(* CODESYS project TrabalhoFMSSFC.project

Project tree, tasks and I/O mapping:
  Device : CODESYS Control Win V3, 3S - Smart Software Solutions GmbH, order no. 305021, version 3.5.11.30
    application Application
      libraries: Standard, * (System)
      task MainTask (cyclic, interval t#20ms, priority 1) calls Inicializacao
      program Inicializacao [SFC]
      program estacaoPallet [SFC]
      program SaidaPecas [SFC]
      program esteira [SFC]
      program RobosDaora [SFC]
      program EstacaoTampa [SFC]
      program Armazenamento [SFC]
  program Inicializacao [SFC]
  program POU [CFC]
*)

// Device/Application/Inicializacao
PROGRAM Inicializacao
VAR
	Bot: INT;
	o_lig: INT;
	o_off: INT;
	o_On: INT;
	Botao_on: BOOL;
	Botao_off: BOOL;
END_VAR

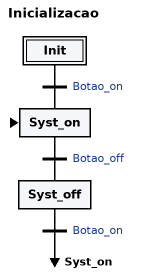
INITIAL_STEP Init:
END_STEP
TRANSITION FROM Init TO Syst_on
    := Botao_on;
END_TRANSITION
STEP Syst_on:
END_STEP
TRANSITION FROM Syst_on TO Syst_off
    := Botao_off;
END_TRANSITION
STEP Syst_off:
END_STEP
TRANSITION FROM Syst_off TO Syst_on
    := Botao_on;
END_TRANSITION

END_PROGRAM

// Inicializacao
PROGRAM Inicializacao
VAR
	Bot: INT;
	o_lig: INT;
	o_off: INT;
	o_On: INT;
	Botao_on: BOOL;
	Botao_off: BOOL;
END_VAR

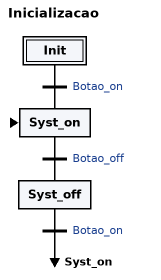
INITIAL_STEP Init:
END_STEP
TRANSITION FROM Init TO Syst_on
    := Botao_on;
END_TRANSITION
STEP Syst_on:
END_STEP
TRANSITION FROM Syst_on TO Syst_off
    := Botao_off;
END_TRANSITION
STEP Syst_off:
END_STEP
TRANSITION FROM Syst_off TO Syst_on
    := Botao_on;
END_TRANSITION

END_PROGRAM

// Device/Application/estacaoPallet
PROGRAM estacaoPallet
VAR_INPUT
END_VAR
VAR_OUTPUT
END_VAR
VAR
	Sistema_on: BOOL;
	diffuse_sensor_3_clp: BOOL;
	diffuse_sensor_4_clp: BOOL;
	timer_1: BOOL;
	timer_2: BOOL;
	timer_3: BOOL;
	timer_5: BOOL;
	timer_6: BOOL;
	timer_7: BOOL;
	timer_8: BOOL;
	timer_9: BOOL;
END_VAR

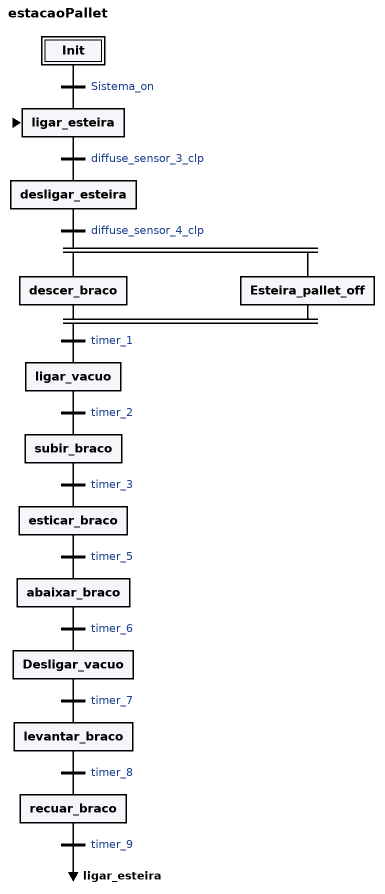
INITIAL_STEP Init:
END_STEP
TRANSITION FROM Init TO ligar_esteira
    := Sistema_on;
END_TRANSITION
STEP ligar_esteira:
END_STEP
TRANSITION FROM ligar_esteira TO desligar_esteira
    := diffuse_sensor_3_clp;
END_TRANSITION
STEP desligar_esteira:
END_STEP
TRANSITION FROM desligar_esteira TO (descer_braco, Esteira_pallet_off)
    := diffuse_sensor_4_clp;
END_TRANSITION
STEP descer_braco:
END_STEP
STEP Esteira_pallet_off:
END_STEP
TRANSITION FROM (descer_braco, Esteira_pallet_off) TO ligar_vacuo
    := timer_1;
END_TRANSITION
STEP ligar_vacuo:
END_STEP
TRANSITION FROM ligar_vacuo TO subir_braco
    := timer_2;
END_TRANSITION
STEP subir_braco:
END_STEP
TRANSITION FROM subir_braco TO esticar_braco
    := timer_3;
END_TRANSITION
STEP esticar_braco:
END_STEP
TRANSITION FROM esticar_braco TO abaixar_braco
    := timer_5;
END_TRANSITION
STEP abaixar_braco:
END_STEP
TRANSITION FROM abaixar_braco TO Desligar_vacuo
    := timer_6;
END_TRANSITION
STEP Desligar_vacuo:
END_STEP
TRANSITION FROM Desligar_vacuo TO levantar_braco
    := timer_7;
END_TRANSITION
STEP levantar_braco:
END_STEP
TRANSITION FROM levantar_braco TO recuar_braco
    := timer_8;
END_TRANSITION
STEP recuar_braco:
END_STEP
TRANSITION FROM recuar_braco TO ligar_esteira
    := timer_9;
END_TRANSITION

END_PROGRAM

// POU
PROGRAM POU
VAR
END_VAR

END_PROGRAM

// Device/Application/SaidaPecas
PROGRAM SaidaPecas
VAR
	Sist_on: BOOL;
	sensor_back: BOOL;
	sensor_front: BOOL;
	azul: BOOL;
	timer_1: BOOL;
	timer_2: BOOL;
	nao_azul: BOOL;
	zera_azul: BOOL;
END_VAR

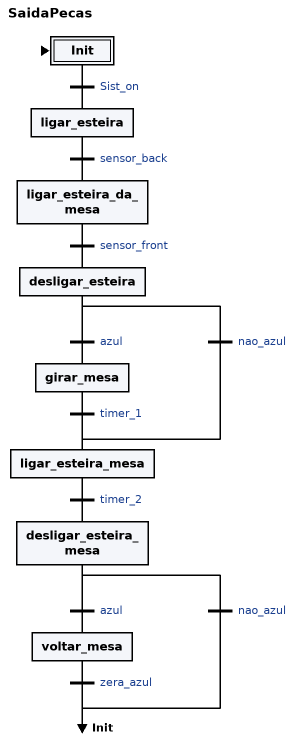
INITIAL_STEP Init:
END_STEP
TRANSITION FROM Init TO ligar_esteira
    := Sist_on;
END_TRANSITION
STEP ligar_esteira:
END_STEP
TRANSITION FROM ligar_esteira TO ligar_esteira_da_mesa
    := sensor_back;
END_TRANSITION
STEP ligar_esteira_da_mesa:
END_STEP
TRANSITION FROM ligar_esteira_da_mesa TO desligar_esteira
    := sensor_front;
END_TRANSITION
STEP desligar_esteira:
END_STEP
TRANSITION FROM desligar_esteira TO girar_mesa
    := azul;
END_TRANSITION
STEP girar_mesa:
END_STEP
TRANSITION FROM girar_mesa TO ligar_esteira_mesa
    := timer_1;
END_TRANSITION
TRANSITION FROM desligar_esteira TO ligar_esteira_mesa
    := nao_azul;
END_TRANSITION
STEP ligar_esteira_mesa:
END_STEP
TRANSITION FROM ligar_esteira_mesa TO desligar_esteira_mesa
    := timer_2;
END_TRANSITION
STEP desligar_esteira_mesa:
END_STEP
TRANSITION FROM desligar_esteira_mesa TO voltar_mesa
    := azul;
END_TRANSITION
STEP voltar_mesa:
END_STEP
TRANSITION FROM voltar_mesa TO Init
    := zera_azul;
END_TRANSITION
TRANSITION FROM desligar_esteira_mesa TO Init
    := nao_azul;
END_TRANSITION

END_PROGRAM

// Device/Application/esteira
PROGRAM esteira
VAR
	Bot: INT;
	o_lig: INT;
	o_off: INT;
	o_On: INT;
	Botao_on: BOOL;
	Botao_off: BOOL;
	Sensor_on: BOOL;
	Sensor_pff: BOOL;
	Sensor_off: BOOL;
	Sensor_Dif: BOOL;
	Sensor_Verde_on: BOOL;
	Sensor_Verde_off: BOOL;
	Timer_on: BOOL;
	Timer1_off: BOOL;
	Timer1_on: BOOL;
	Reset_Blade: BOOL;
	Sensor_presenca: BOOL;
	Sensor_Dif_on: BOOL;
	Sensor_Dif_off: BOOL;
	End_Blade: BOOL;
	Sensor_Dif1_on: BOOL;
	Sensor_Dif1_off: BOOL;
END_VAR

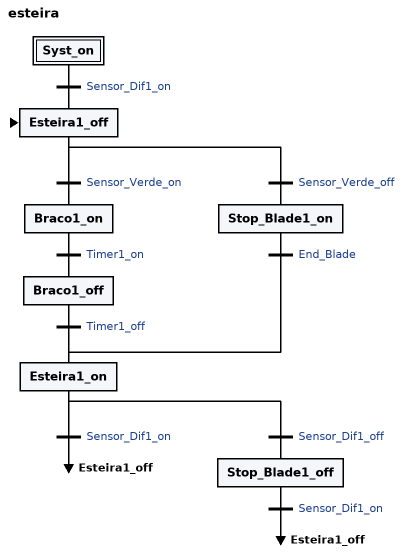
INITIAL_STEP Syst_on:
END_STEP
TRANSITION FROM Syst_on TO Esteira1_off
    := Sensor_Dif1_on;
END_TRANSITION
STEP Esteira1_off:
END_STEP
TRANSITION FROM Esteira1_off TO Braco1_on
    := Sensor_Verde_on;
END_TRANSITION
STEP Braco1_on:
END_STEP
TRANSITION FROM Braco1_on TO Braco1_off
    := Timer1_on;
END_TRANSITION
STEP Braco1_off:
END_STEP
TRANSITION FROM Braco1_off TO Esteira1_on
    := Timer1_off;
END_TRANSITION
TRANSITION FROM Esteira1_off TO Stop_Blade1_on
    := Sensor_Verde_off;
END_TRANSITION
STEP Stop_Blade1_on:
END_STEP
TRANSITION FROM Stop_Blade1_on TO Esteira1_on
    := End_Blade;
END_TRANSITION
STEP Esteira1_on:
END_STEP
TRANSITION FROM Esteira1_on TO Esteira1_off
    := Sensor_Dif1_on;
END_TRANSITION
TRANSITION FROM Esteira1_on TO Stop_Blade1_off
    := Sensor_Dif1_off;
END_TRANSITION
STEP Stop_Blade1_off:
END_STEP
TRANSITION FROM Stop_Blade1_off TO Esteira1_off
    := Sensor_Dif1_on;
END_TRANSITION

END_PROGRAM

// Device/Application/RobosDaora
PROGRAM RobosDaora
VAR
	Bot: INT;
	o_lig: INT;
	o_off: INT;
	o_On: INT;
	Botao_on: BOOL;
	Botao_off: BOOL;
	Robo1_Sens: BOOL;
	Robo1_Sens_on: BOOL;
	Robo1_end: BOOL;
END_VAR

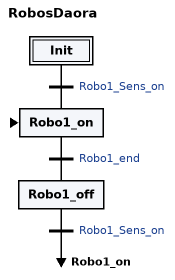
INITIAL_STEP Init:
END_STEP
TRANSITION FROM Init TO Robo1_on
    := Robo1_Sens_on;
END_TRANSITION
STEP Robo1_on:
END_STEP
TRANSITION FROM Robo1_on TO Robo1_off
    := Robo1_end;
END_TRANSITION
STEP Robo1_off:
END_STEP
TRANSITION FROM Robo1_off TO Robo1_on
    := Robo1_Sens_on;
END_TRANSITION

END_PROGRAM

// Device/Application/EstacaoTampa
PROGRAM EstacaoTampa
VAR
	//Entradas
	VisionSensor4_1:BOOL;
	VisionSensor4_0:BOOL;
	VIsionSensor4_2:BOOL;
	//SAIDAS
	Conveyor2m3:BOOL;
	PosicaoPegar: BOOL;
	ZPosition: BOOL;
	BoxDetected: BOOL;
	Grabber: BOOL;
	TampaPega: BOOL;
	Timer1: BOOL;
	Timer2: BOOL;
	PosicaoTampar: BOOL;
	Timer3: BOOL;
	Timer4: BOOL;
	Timer5: BOOL;
	StopBlade: BOOL;
	VisionSensor4_1Negado: BOOL;
END_VAR

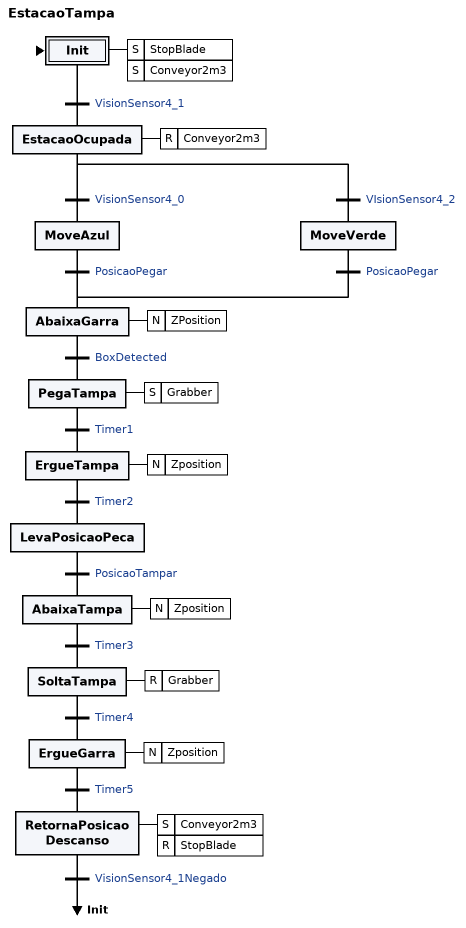
INITIAL_STEP Init:
    StopBlade(S);
    Conveyor2m3(S);
END_STEP
TRANSITION FROM Init TO EstacaoOcupada
    := VisionSensor4_1;
END_TRANSITION
STEP EstacaoOcupada:
    Conveyor2m3(R);
END_STEP
TRANSITION FROM EstacaoOcupada TO MoveAzul
    := VisionSensor4_0;
END_TRANSITION
STEP MoveAzul:
END_STEP
TRANSITION FROM MoveAzul TO AbaixaGarra
    := PosicaoPegar;
END_TRANSITION
TRANSITION FROM EstacaoOcupada TO MoveVerde
    := VIsionSensor4_2;
END_TRANSITION
STEP MoveVerde:
END_STEP
TRANSITION FROM MoveVerde TO AbaixaGarra
    := PosicaoPegar;
END_TRANSITION
STEP AbaixaGarra:
    ZPosition(N);
END_STEP
TRANSITION FROM AbaixaGarra TO PegaTampa
    := BoxDetected;
END_TRANSITION
STEP PegaTampa:
    Grabber(S);
END_STEP
TRANSITION FROM PegaTampa TO ErgueTampa
    := Timer1;
END_TRANSITION
STEP ErgueTampa:
    Zposition(N);
END_STEP
TRANSITION FROM ErgueTampa TO LevaPosicaoPeca
    := Timer2;
END_TRANSITION
STEP LevaPosicaoPeca:
END_STEP
TRANSITION FROM LevaPosicaoPeca TO AbaixaTampa
    := PosicaoTampar;
END_TRANSITION
STEP AbaixaTampa:
    Zposition(N);
END_STEP
TRANSITION FROM AbaixaTampa TO SoltaTampa
    := Timer3;
END_TRANSITION
STEP SoltaTampa:
    Grabber(R);
END_STEP
TRANSITION FROM SoltaTampa TO ErgueGarra
    := Timer4;
END_TRANSITION
STEP ErgueGarra:
    Zposition(N);
END_STEP
TRANSITION FROM ErgueGarra TO RetornaPosicaoDescanso
    := Timer5;
END_TRANSITION
STEP RetornaPosicaoDescanso:
    Conveyor2m3(S);
    StopBlade(R);
END_STEP
TRANSITION FROM RetornaPosicaoDescanso TO Init
    := VisionSensor4_1Negado;
END_TRANSITION

END_PROGRAM

// Device/Application/Armazenamento
PROGRAM Armazenamento
VAR
	At_Load: BOOL;
	Timer_1: BOOL;
	Timer_2: BOOL;
	Timer_3: BOOL;
	Timer_4: BOOL;
	Timer_5: BOOL;
	Timer_6: BOOL;
	Timer_7: BOOL;
	Timer_0: BOOL;
	Timer_8: BOOL;
	teste: BOOL;
	timer_9: BOOL;
	Timer_10: BOOL;
	Timer_11: BOOL;
	Timer_12: BOOL;
	Timer_13: BOOL;
	Timer_14: BOOL;
	Timer_15: BOOL;
	Timer_16: BOOL;
END_VAR

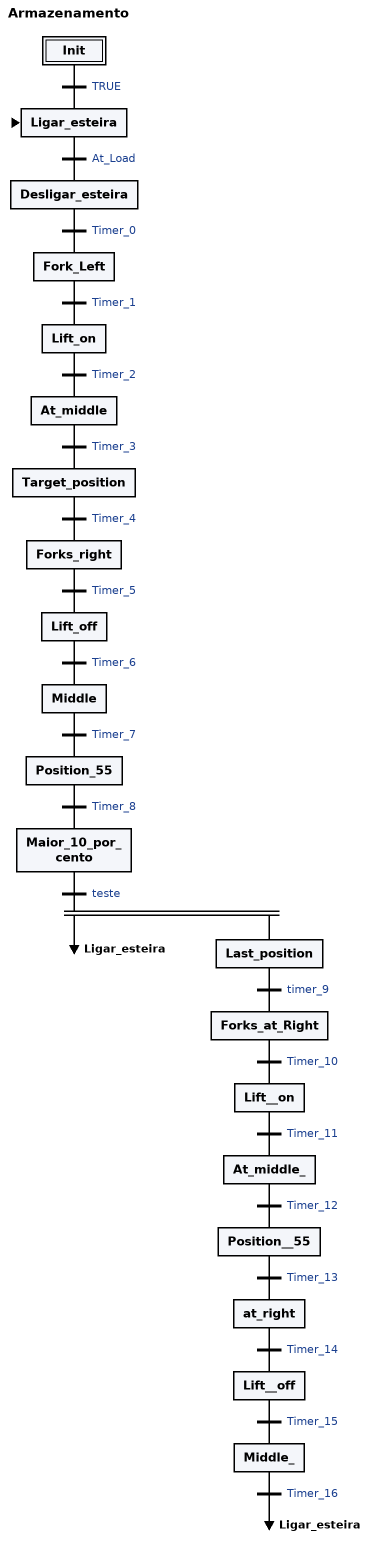
INITIAL_STEP Init:
END_STEP
TRANSITION FROM Init TO Ligar_esteira
    := TRUE;
END_TRANSITION
STEP Ligar_esteira:
END_STEP
TRANSITION FROM Ligar_esteira TO Desligar_esteira
    := At_Load;
END_TRANSITION
STEP Desligar_esteira:
END_STEP
TRANSITION FROM Desligar_esteira TO Fork_Left
    := Timer_0;
END_TRANSITION
STEP Fork_Left:
END_STEP
TRANSITION FROM Fork_Left TO Lift_on
    := Timer_1;
END_TRANSITION
STEP Lift_on:
END_STEP
TRANSITION FROM Lift_on TO At_middle
    := Timer_2;
END_TRANSITION
STEP At_middle:
END_STEP
TRANSITION FROM At_middle TO Target_position
    := Timer_3;
END_TRANSITION
STEP Target_position:
END_STEP
TRANSITION FROM Target_position TO Forks_right
    := Timer_4;
END_TRANSITION
STEP Forks_right:
END_STEP
TRANSITION FROM Forks_right TO Lift_off
    := Timer_5;
END_TRANSITION
STEP Lift_off:
END_STEP
TRANSITION FROM Lift_off TO Middle
    := Timer_6;
END_TRANSITION
STEP Middle:
END_STEP
TRANSITION FROM Middle TO Position_55
    := Timer_7;
END_TRANSITION
STEP Position_55:
END_STEP
TRANSITION FROM Position_55 TO Maior_10_por_cento
    := Timer_8;
END_TRANSITION
STEP Maior_10_por_cento:
END_STEP
TRANSITION FROM Maior_10_por_cento TO (Ligar_esteira, Last_position)
    := teste;
END_TRANSITION
STEP Last_position:
END_STEP
TRANSITION FROM Last_position TO Forks_at_Right
    := timer_9;
END_TRANSITION
STEP Forks_at_Right:
END_STEP
TRANSITION FROM Forks_at_Right TO Lift__on
    := Timer_10;
END_TRANSITION
STEP Lift__on:
END_STEP
TRANSITION FROM Lift__on TO At_middle_
    := Timer_11;
END_TRANSITION
STEP At_middle_:
END_STEP
TRANSITION FROM At_middle_ TO Position__55
    := Timer_12;
END_TRANSITION
STEP Position__55:
END_STEP
TRANSITION FROM Position__55 TO at_right
    := Timer_13;
END_TRANSITION
STEP at_right:
END_STEP
TRANSITION FROM at_right TO Lift__off
    := Timer_14;
END_TRANSITION
STEP Lift__off:
END_STEP
TRANSITION FROM Lift__off TO Middle_
    := Timer_15;
END_TRANSITION
STEP Middle_:
END_STEP
TRANSITION FROM Middle_ TO Ligar_esteira
    := Timer_16;
END_TRANSITION

END_PROGRAM
